Yaskawa INFORM job: FRONT_SEARCH_-90ST-1_4940TEST1.JBI

/JOB
//NAME FRONT_SEARCH_-90ST-1_4940TEST1
//POS
///NPOS 28,28,0,6,0,0
///TOOL 0
///POSTYPE PULSE
///PULSE
C00000=23,-11312,44619,-84866,32848,-77368
///LIMIT ON
C00001=-42517,-20143,9725,-37936,102,56716
///LIMIT OFF
C00002=-54051,-18376,-3566,35720,24131,28196
C00003=-52287,-12134,7109,37600,21316,27372
C00004=-51932,-10734,9554,38203,20680,27100
C00005=-51067,-9690,10529,37015,20415,27772
C00006=-51291,-9073,12879,39225,19611,26646
C00007=-51932,-10734,9554,38203,20680,27100
///LIMIT ON
C00008=-18684,-22097,1147,-186475,-11922,-28191
C00009=-18684,-22097,1147,-186475,-11922,-28191
C00010=-18505,-21432,1640,-186682,-12099,-28079
C00011=-18610,-20693,4284,-187745,-10854,-27577
C00012=-18684,-22097,1147,-186475,-11922,-28191
///LIMIT OFF
C00013=17491,-23321,-3623,-46801,26124,78240
C00014=17491,-23321,-3623,-46801,26124,78240
C00015=17208,-22413,-2956,-46274,26135,77937
C00016=17303,-21930,-919,-47894,25495,78796
C00017=17491,-23321,-3623,-46801,26124,78240
C00018=19665,-34863,-16820,-49823,29128,-29934
///LIMIT ON
C00019=20305,-24307,-1379,-197886,-11660,35857
C00020=19862,-24323,-795,-197520,-11164,35639
C00021=19487,-23341,-100,-196010,-11310,34880
C00022=19600,-22857,1827,-198244,-10452,35959
C00023=19862,-24323,-795,-197520,-11164,35639
C00024=23011,-43288,-23551,-202387,-13314,38280
///LIMIT OFF
C00025=53387,-41933,-2884,-72369,37540,-39448
C00026=-706,-35551,42177,34860,-9217,2477
C00027=262,-52278,40443,-360,6873,247
BC00000=843729
BC00001=939330
BC00002=939330
BC00003=939330
BC00004=939330
BC00005=939330
BC00006=939330
BC00007=939330
BC00008=939331
BC00009=939331
BC00010=939331
BC00011=939331
BC00012=939331
BC00013=939330
BC00014=939330
BC00015=939330
BC00016=939330
BC00017=939330
BC00018=939330
BC00019=939330
BC00020=939330
BC00021=939330
BC00022=939330
BC00023=939330
BC00024=925964
BC00025=880626
BC00026=766275
BC00027=759398
///POSTYPE BASE
///RECTAN
///RCONF 0,0,0,0,0,0,0,0,0,0,0,0,0,0,0,0,0,0,0,0,0,0,0,0
P00006=-2.449,0.031,8.825,0.0000,0.0000,0.0000
P00058=0.000,0.000,3.000,0.0000,0.0000,0.0000
P00501=-2.026,0.009,3.534,0.0000,0.0000,0.0000
///RCONF 1,0,0,0,0,0,0,0,0,0,0,0,0,0,0,0,0,0,0,0,0,0,0,0
P00502=-2.023,0.001,1.732,0.0000,0.0000,0.0000
P00503=0.138,-0.044,1.539,0.0000,0.0000,0.0000
P00504=-0.309,-0.010,1.636,0.0000,0.0000,0.0000
//INST
///DATE 2024/06/12 15:16
///ATTR SC,RW
///GROUP1 RB1,BS1
NOP
MOVJ C00000 BC00000 VJ=40.00
'::::::::::::::::::::::::::::::::
'W56 P
'::::::::::::::::::::::::::::::::
MOVL C00001 BC00001 V=500.0
MOVL C00002 BC00002 V=500.0
MOVL C00003 BC00003 V=500.0
MOVL C00004 BC00004 V=166.7 PL=0
REFP 3 C00005 BC00005
CALL JOB:SEARCH-R1
IMOV P0058 V=23.0
SET P0501 P0006
SFTON P0501
REFP 3 C00006 BC00006
CALL JOB:SEARCH-R1
SET P0501 P0006
SFTON P0501
MOVL C00007 BC00007 V=166.7 PL=0
SFTOF
'::::::::::::::::::::::::::::::::
'W56 L
'::::::::::::::::::::::::::::::::
MOVL C00008 BC00008 V=333.3
MOVL C00009 BC00009 V=166.7 PL=0
REFP 3 C00010 BC00010
CALL JOB:SEARCH-R1
IMOV P0058 V=23.0
SET P0502 P0006
SFTON P0502
REFP 3 C00011 BC00011
CALL JOB:SEARCH-R1
SET P0502 P0006
SFTON P0502
MOVL C00012 BC00012 V=166.7 PL=0
SFTOF
'::::::::::::::::::::::::::::::::
'W57 P
'::::::::::::::::::::::::::::::::
MOVL C00013 BC00013 V=250.0
MOVL C00014 BC00014 V=166.7 PL=0
REFP 3 C00015 BC00015
CALL JOB:SEARCH-R1
IMOV P0058 V=23.0
SET P0503 P0006
SFTON P0503
REFP 3 C00016 BC00016
CALL JOB:SEARCH-R1
SET P0503 P0006
SFTON P0503
MOVL C00017 BC00017 V=250.0 PL=0
SFTOF
'::::::::::::::::::::::::::::::::
'W57 L
'::::::::::::::::::::::::::::::::
MOVL C00018 BC00018 V=333.3
MOVL C00019 BC00019 V=333.3
MOVL C00020 BC00020 V=166.7 PL=0
REFP 3 C00021 BC00021
CALL JOB:SEARCH-R1
IMOV P0058 V=23.0
SET P0504 P0006
SFTON P0504
REFP 3 C00022 BC00022
CALL JOB:SEARCH-R1
SET P0504 P0006
SFTON P0504
MOVL C00023 BC00023 V=166.7 PL=0
SFTOF
MOVJ C00024 BC00024 VJ=40.00
MOVJ C00025 BC00025 VJ=50.00
MOVJ C00026 BC00026 VJ=50.00
MOVJ C00027 BC00027 VJ=50.00
END
